// TIA Portal V18 export
DATA_BLOCK "03_FDBACK"   // DB5, F_DB
{ S7_Optimized_Access := 'TRUE'; DB_Accessible_From_OPC_UA := 'FALSE' }
// stored: DBAccessibleFromOPCUA false
   VAR
      AlwaysFALSE : Bool;
      AlwaysTRUE : Bool := TRUE;
      "!!ITERATOR_STRINGS$$" : Bool;
      "!!03_FDBACK.{db_element}$$" : Bool;
   END_VAR
BEGIN
END_DATA_BLOCK
